TYPE ST_ACDCCharger_params :
STRUCT
	b_ACDCChargerFitted		:	BOOL;
	ui_NrOfInstalledModules	:	UINT	:=	2;
	ui_ModuleDesignPower	:	Uint	:=	30;
	r_VoltageWindow			:	REAL	:=  2;
	GridVoltageHysteresis	: 	REAL	:=	2;
	BMSChargeLimitRampRate	:	REAL	:=	0.5; //DC amps per cycle;
	SocHysteresis			:	Real	:=	2;
END_STRUCT
END_TYPE

(* stored: Version 1.1.0.1, ProductVersion 3.1.4026.18
   DUT ST_ACDCCharger_params: Id {dc3f54bf-c14a-4b40-824d-6bf22d577d68} *)
